// TIA Portal V19 export
VAR_GLOBAL   // PLC tag table "Default tag table"
   System_Byte AT %MB1 : Byte;
   FirstScan AT %M1.0 : Bool;
   DiagStatusUpdate AT %M1.1 : Bool;
   AlwaysTRUE AT %M1.2 : Bool;
   AlwaysFALSE AT %M1.3 : Bool;
   Clock_Byte AT %MB0 : Byte;
   Clock_10Hz AT %M0.0 : Bool;
   Clock_5Hz AT %M0.1 : Bool;
   "Clock_2.5Hz" AT %M0.2 : Bool;
   Clock_2Hz AT %M0.3 : Bool;
   "Clock_1.25Hz" AT %M0.4 : Bool;
   Clock_1Hz AT %M0.5 : Bool;
   "Clock_0.625Hz" AT %M0.6 : Bool;
   "Clock_0.5Hz" AT %M0.7 : Bool;
   "MGF FEED PUMP W/S" AT %I24.4 : Bool;
   "RO FEED PUMP W/S" AT %I24.5 : Bool;
   "RO HPP PUMP W/S" AT %I24.6 : Bool;
   "LS-10 HIGH" AT %I24.7 : Bool;
   "regenration process  start" AT %M2.1 : Bool;
   "test bit trail" AT %M2.0 : Bool;
   JJJ AT %M2.2 : Bool;
   III AT %M2.3 : Bool;
   QQQ AT %M2.4 : Bool;
END_VAR
